// Unit host for the §6.12 parallel suite: two children, one forking chain.
FUNCTION_BLOCK FB_ProbeUnitPar EXTENDS FB_UnitBase
VAR
    ChildA : FB_ProbeCM;
    ChildB : FB_ProbeCM;
    Chain : FB_ProbeParChain;
END_VAR

Cyclic();

METHOD Setup : BOOL
VAR_INPUT
    Name : STRING(80);
END_VAR
_M_SetName(Name);
StallTime := T#10S;
Setup := ChildA.Setup(Name := CONCAT(Name, '.ChildA'))
    AND ChildB.Setup(Name := CONCAT(Name, '.ChildB'))
    AND _M_Register(Child := ChildA)
    AND _M_Register(Child := ChildB)
    AND Chain.Setup(Host := THIS^, ChildA := ChildA, ChildB := ChildB);
END_METHOD

METHOD PROTECTED OnCyclic : DINT
OnCyclic := SUPER^.OnCyclic();   // base first (Core §3.14.2)
_M_TickChildren();
END_METHOD

METHOD PROTECTED _M_Dispatch
Chain.M_Run();
END_METHOD

METHOD PROTECTED OnCommandStart : DINT
OnCommandStart := SUPER^.OnCommandStart();
Chain.M_Reset();
END_METHOD

METHOD M_TestSetChild : BOOL
VAR_INPUT
    Which : INT;
    ChildDone : BOOL;
END_VAR
IF Which = 1 THEN
    ChildA.SimDone := ChildDone;
ELSE
    ChildB.SimDone := ChildDone;
END_IF
M_TestSetChild := TRUE;
END_METHOD

METHOD M_TestIssues : UDINT
VAR_INPUT
    Leg : INT;
END_VAR
M_TestIssues := Chain.M_TestIssues(Leg := Leg);
END_METHOD

METHOD M_TestChainStep : INT
M_TestChainStep := Chain.ActiveStep;
END_METHOD

END_FUNCTION_BLOCK

(* stored: Version 1.1.0.1, ProductVersion 3.1.4024.12
   POU FB_ProbeUnitPar: Id {ae9fb4ff-77d4-4a3b-ad12-a290eb4c0e93}, SpecialFunc None
   Method Setup: Id {5529537b-a583-43f3-bce8-f173ea5e9a6e}
   Method OnCyclic: Id {35120a6e-e494-4830-9cd1-221ad5fa8a76}
   Method _M_Dispatch: Id {bca17faf-c3ab-4478-bfaf-f89487af1efc}
   Method OnCommandStart: Id {231ee97c-b4fe-426f-8940-65d5066fed47}
   Method M_TestSetChild: Id {332e50ad-63c4-4a09-be6f-efd65326a0e8}
   Method M_TestIssues: Id {8b66b073-547b-47f4-8ee3-2a8c191daa0f}
   Method M_TestChainStep: Id {ecb1c3f2-972e-481d-b614-1b07cbb06a46} *)
